INTERFACE I_NodePrototypeVisitor

METHOD VisitNodePrototype
VAR_INPUT
	VisitingPrototype : I_NodePrototype;
END_VAR
END_METHOD

END_INTERFACE

(* stored: Version 1.1.0.1, ProductVersion 3.1.4024.12
   Itf I_NodePrototypeVisitor: Id {15e4ba15-5e09-07af-1d62-3fd10eef8bb9}
   Method VisitNodePrototype: Id {d384a963-8323-0952-0376-8fbe4c7b2e5e} *)
